FUNCTION_BLOCK ScriblySequenceStop EXTENDS ScriblySequence IMPLEMENTS ZCore.ISequence
VAR
  _step : ZCore.Step(ScriblyStep.StopBegin, ScriblyStep.StopEnd);
  _timerSim : ZAux.Timer;
END_VAR

IF OnStart(_step) THEN
  ; // init custom sequence variables here ...
END_IF

REPEAT
  LogStep();

  CASE _step.Index OF
    (* -------------------------------------------------------------------------------------------------------------------------------- *)
    ScriblyStep.StopBegin:
    (* -------------------------------------------------------------------------------------------------------------------------------- *)
      IF _step.OnEntry()
      THEN
        _timerSim.WaitAsync(5);
			END_IF
      
      Await(_timerSim, nextStep:=ScriblyStep.StopEnd);
      // _step.SetNext(index:=ScriblyStep.StopEnd);

    (* -------------------------------------------------------------------------------------------------------------------------------- *)
    ScriblyStep.StopEnd:
    (* -------------------------------------------------------------------------------------------------------------------------------- *)    
      SetBusy(FALSE);
  
  ELSE
    Abort('sequence contains unhandled step');
  END_CASE
UNTIL _step.IsNotRepeatable() OR_ELSE NOT Busy END_REPEAT

END_FUNCTION_BLOCK

(* stored: Version 1.1.0.1
   POU ScriblySequenceStop: Id {7d641f4f-31b2-4693-b78a-d201a83e91aa}, SpecialFunc None *)
